SUBAPPLICATION Versuch_403 (* Versuch Array Summe *)
  (* Standard: 61499-2; Description: Copyright (c) 2023 Meisterschulen am Ostbahnhof This program and the accompanying materials are made available under the terms of the Eclipse Public License 2.0 which is available at https://www.eclipse.org/legal/epl-2.0/ SPDX-License-Identifier: EPL-2.0 *)
  (* Version 1.0, 2023-10-23, Franz Höpfinger, Meisterschulen am Ostbahnhof, initial API and implementation and/or initial documentation *)
  PACKAGE Versuche;
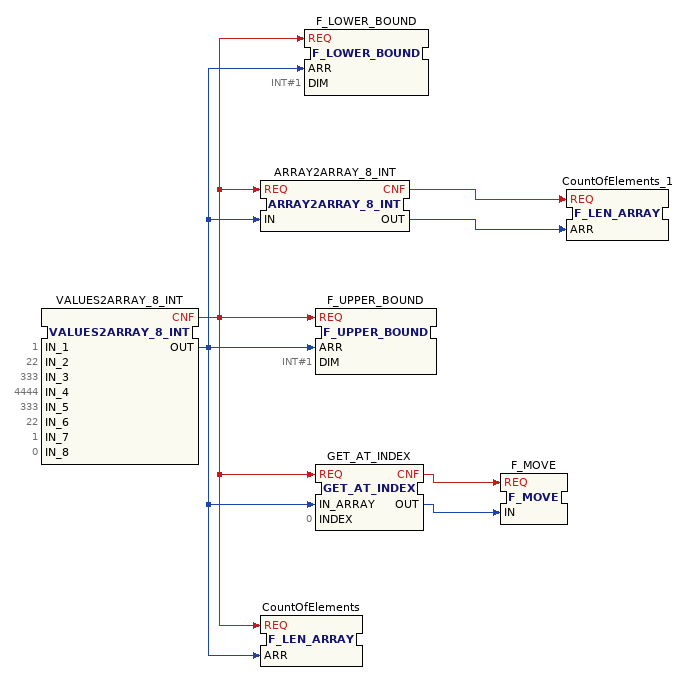
  FBS
    GET_AT_INDEX : eclipse4diac::convert::GET_AT_INDEX(INDEX := 0);
    F_MOVE : iec61131::selection::F_MOVE; {SET_ATTRIBUTE(DataType, INT)}
    CountOfElements : eclipse4diac::utils::arrays::F_LEN_ARRAY;
    F_UPPER_BOUND : iec61131::arrays::F_UPPER_BOUND(DIM := INT#1);
    F_LOWER_BOUND : iec61131::arrays::F_LOWER_BOUND(DIM := INT#1);
    VALUES2ARRAY_8_INT : eclipse4diac::convert::VALUES2ARRAY_8_INT(IN_1 := 1, IN_2 := 22, IN_3 := 333, IN_4 := 4444, IN_5 := 333, IN_6 := 22, IN_7 := 1, IN_8 := 0);
    ARRAY2ARRAY_8_INT : eclipse4diac::convert::ARRAY2ARRAY_8_INT;
    CountOfElements_1 : eclipse4diac::utils::arrays::F_LEN_ARRAY;
  END_FBS
  EVENT_CONNECTIONS
    GET_AT_INDEX.CNF TO F_MOVE.REQ;
    VALUES2ARRAY_8_INT.CNF TO GET_AT_INDEX.REQ;
    VALUES2ARRAY_8_INT.CNF TO CountOfElements.REQ;
    VALUES2ARRAY_8_INT.CNF TO F_LOWER_BOUND.REQ;
    VALUES2ARRAY_8_INT.CNF TO F_UPPER_BOUND.REQ;
    VALUES2ARRAY_8_INT.CNF TO ARRAY2ARRAY_8_INT.REQ;
    ARRAY2ARRAY_8_INT.CNF TO CountOfElements_1.REQ;
  END_CONNECTIONS
  DATA_CONNECTIONS
    GET_AT_INDEX.OUT TO F_MOVE.IN;
    VALUES2ARRAY_8_INT.OUT TO GET_AT_INDEX.IN_ARRAY;
    VALUES2ARRAY_8_INT.OUT TO F_UPPER_BOUND.ARR;
    VALUES2ARRAY_8_INT.OUT TO F_LOWER_BOUND.ARR;
    VALUES2ARRAY_8_INT.OUT TO CountOfElements.ARR;
    VALUES2ARRAY_8_INT.OUT TO ARRAY2ARRAY_8_INT.IN;
    ARRAY2ARRAY_8_INT.OUT TO CountOfElements_1.ARR;
  END_CONNECTIONS
END_SUBAPPLICATION
